Yaskawa INFORM job: PARK-POS-ZONE-1-AUTO.JBI

/JOB
//NAME PARK-POS-ZONE-1-AUTO
//POS
///NPOS 1,1,0,0,0,0
///TOOL 0
///POSTYPE PULSE
///PULSE
C00000=-100644,-58707,-30728,26719,55125,30643
BC00000=208121
//INST
///DATE 2018/10/02 16:06
///ATTR SC,RW
///GROUP1 RB1,BS1
NOP
SFTOF
MOVJ C00000 BC00000 VJ=20.00
END
